/// machine data that is used through most sequences of the unit (motor speed, axes positions, ...)
TYPE QualityInspectionDataMachine :
STRUCT
  Slowspeed : LREAL;
  Highspeed : LREAL;
END_STRUCT
END_TYPE

(* stored: Version 1.1.0.1
   DUT QualityInspectionDataMachine: Id {d9362f81-57b2-4524-9fa0-d35d64e42a26} *)
